TYPE LAxisCtrl_typeTorqueLimiting :
STRUCT

	TorqueLimit	: LREAL;
	mode			: DINT;

END_STRUCT
END_TYPE

(* stored: Version 1.1.0.1
   DUT LAxisCtrl_typeTorqueLimiting: Id {dc0876e8-a04d-45bd-8d87-d42eebe0ab36} *)
